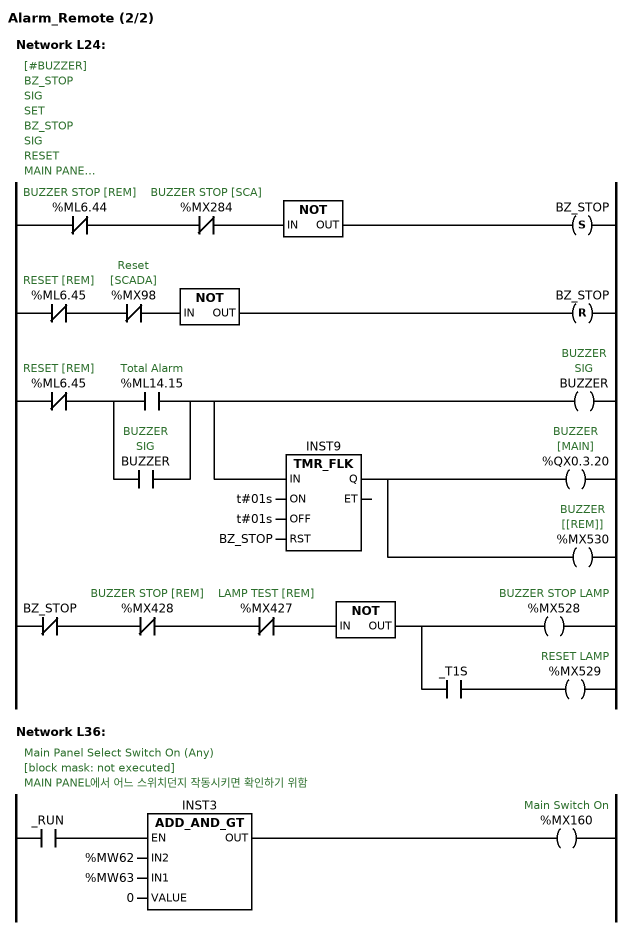
(* [picture p24: Alarm_Remote rungs L24-L36] *)
(* [#BUZZER] *)
(* Rung L24 *)
IF NOT (NOT %ML6.44 AND NOT %MX284) THEN BZ_STOP := TRUE; END_IF;
IF NOT (NOT %ML6.45 AND NOT %MX98) THEN BZ_STOP := FALSE; END_IF;
_p1 := NOT %ML6.45 AND (%ML14.15 OR BUZZER);
BUZZER := _p1;
INST9(IN := _p1, ON := t#01s, OFF := t#01s, RST := BZ_STOP);
%QX0.3.20 := INST9.Q;
%MX530 := INST9.Q;
%MX528 := NOT (NOT BZ_STOP AND NOT %MX428 AND NOT %MX427);
%MX529 := (NOT (NOT BZ_STOP AND NOT %MX428 AND NOT %MX427)) AND _T1S;
(* BZ_STOP / SIG / SET *)
(* BZ_STOP / SIG / RESET *)
(* MAIN PANEL / BUZZER / OUTPUT *)
(* [REM] PANEL / BUZZER / OUTPUT *)
(* Main Panel Select Switch On (Any) *)
(* Rung L36 is block-masked: not executed *)
// IF _RUN THEN INST3(IN2 := %MW62, IN1 := %MW63, VALUE := 0); END_IF;
// %MX160 := INST3.OUT;
(* MAIN PANEL에서 어느 스위치던지 작동시키면 확인하기 위함 *)
END_PROGRAM